(*
SPDX-FileCopyrightText: Â© 2026 Oleksandr Tiutyk <trofimich@gmail.com>
SPDX-License-Identifier: MIT
License: https://opensource.org/license/mit
*)

(*!
<summary>Defines command flags sent from an HMI to an automation component.</summary>
<description>
Command fields are pulsed or set by an operator/HMI interface. The element consumes and resets these flags to FALSE
within its local instance memory upon dispatching the operation.
</description>
*)

TYPE HMI_AUTOMATION_COMPONENT_COMMANDS :
STRUCT
	Enable : BOOL;
	Disable : BOOL;
	
	Reset : BOOL;	
END_STRUCT
END_TYPE

(* stored: Version 1.1.0.1
   DUT HMI_AUTOMATION_COMPONENT_COMMANDS: Id {1590423e-7120-451f-b462-35fc53b7d967} *)
